TYPE ST_StationRecipe :
STRUCT

		Axis			: ST_AxisRecipe;
		//	Travel Time ??
END_STRUCT
END_TYPE

(* stored: Version 1.1.0.1, ProductVersion 3.1.4024.15
   DUT ST_StationRecipe: Id {316f78f7-1d6a-4e87-9088-b3cfa0940815} *)
